// TIA Portal V19 program export: 1 tag tables, 0 data types, 1 data blocks, 3 code blocks (in call order from the OBs), 1 instance data blocks

VAR_GLOBAL   // PLC tag table "Default tag table"
   Tag_1 AT %I0.0 : Bool;
   Tag_2 AT %Q0.0 : Bool;
END_VAR

DATA_BLOCK "Data_block_1"   // DB1
{ S7_Optimized_Access := 'TRUE' }
// stored: MemoryReserve 100
   VAR
      bit1 : Bool;
      bit2 : Bool;
      bit3 : Bool;
      bit4 : Bool;
      bit5 : Bool;
      bit6 : Bool;
      bit7 : Bool;
      bit8 : Bool;
      bit9 : Bool;
      bit10 : Bool;
   END_VAR
BEGIN
END_DATA_BLOCK

ORGANIZATION_BLOCK "Main"   // OB1, LAD, ProgramCycle
TITLE = "Main Program Sweep (Cycle)"
{ S7_Optimized_Access := 'TRUE' }
// stored: SetENOAutomatically false
   VAR_INPUT
      Initial_Call : Bool;   // Initial call of this OB
      Remanence : Bool;   // =True, if remanent data are available
   END_VAR
BEGIN

REGION Network 1: FC call
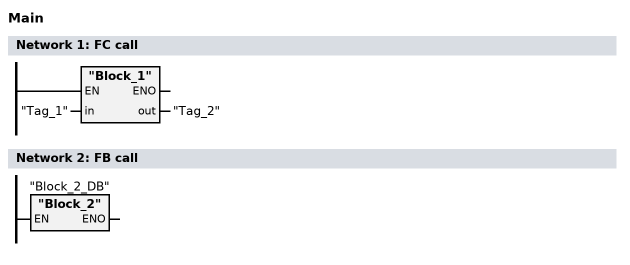
   RUNG wire#powerrail
      "Block_1"(in := "Tag_1", out => "Tag_2")
   END_RUNG
   // the same network as SCL:
   "Block_1"(in := "Tag_1", out => "Tag_2");
END_REGION

REGION Network 2: FB call
   RUNG wire#powerrail
      "Block_2_DB"()
   END_RUNG
   // the same network as SCL:
   "Block_2_DB"();   // "Block_2"
END_REGION
END_ORGANIZATION_BLOCK

FUNCTION "Block_1" : Void   // FC1, FBD
TITLE = FC
{ S7_Optimized_Access := 'TRUE' }
// stored: SetENOAutomatically false
   VAR_INPUT
      in : Bool;
   END_VAR
   VAR_OUTPUT
      out : Bool;
   END_VAR
BEGIN

REGION Network 1: network1
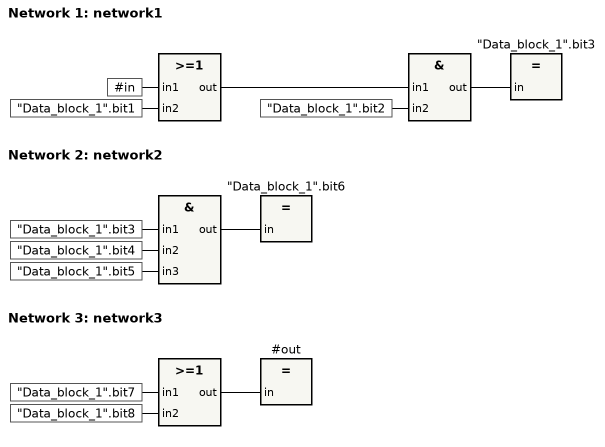
   "Data_block_1".bit3 := (#in OR "Data_block_1".bit1) AND "Data_block_1".bit2;
END_REGION

REGION Network 2: network2
   "Data_block_1".bit6 := "Data_block_1".bit3 AND "Data_block_1".bit4 AND "Data_block_1".bit5;
END_REGION

REGION Network 3: network3
   #out := "Data_block_1".bit7 OR "Data_block_1".bit8;
END_REGION
END_FUNCTION

FUNCTION_BLOCK "Block_2"   // FB1, FBD
TITLE = FB
{ S7_Optimized_Access := 'TRUE' }
// stored: MemoryReserve 100, SetENOAutomatically false
   VAR
      HF : Array[0..10] of Bool;
   END_VAR
BEGIN

REGION Network 1: network 1
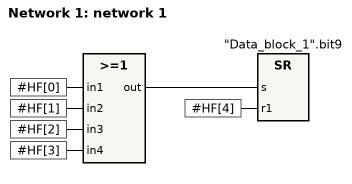
   IF #HF[0] OR #HF[1] OR #HF[2] OR #HF[3] THEN
       "Data_block_1".bit9 := TRUE;   // SR flip-flop
   END_IF;
   IF #HF[4] THEN "Data_block_1".bit9 := FALSE; END_IF;
END_REGION
END_FUNCTION_BLOCK

DATA_BLOCK "Block_2_DB"   // DB2
// stored: InstanceOfName Block_2, InstanceOfType FB
"Block_2"
BEGIN
END_DATA_BLOCK
